Fanuc KAREL source: kf00077.KL

-- PROVISIONAL review KL for V1013-1; original PC SHA256 595889b712698b64770a7bb1107c75c75ea50caefd57440c842ffac2f0f9aed2
-- Incomplete behavior may be omitted. Consult companion uncertainty JSON. Do not deploy.
PROGRAM KF00077
%NOLOCKGROUP
BEGIN
  -- UNRESOLVED_PC offsets 5-15; opcodes 3F,75
  -- UNRESOLVED_PC offsets 20-29; opcodes 3F,75
  -- UNRESOLVED_PC offsets 34-45; opcodes 2E,23
  -- UNRESOLVED_PC offsets 50-61; opcodes 2E,23
  -- UNRESOLVED_PC offsets 66-84; opcodes 27,22,2A,22,31
  -- UNRESOLVED_PC offsets 89-93; opcodes 7F
END KF00077
